// TwinCAT 3 PLC project CX2040_Project
// ProgramVersion: 3.1.4023.0
// libraries:
//   Tc2_EtherCAT, * (Beckhoff Automation GmbH)
//   Tc2_SerialCom, * (Beckhoff Automation GmbH)
//   Tc2_Standard, * (Beckhoff Automation GmbH)
//   Tc2_System, * (Beckhoff Automation GmbH)
//   Tc3_Module, * (Beckhoff Automation GmbH)
// project tree:
//   GVLs/ GVL.TcGVL
//   / PlcTask.TcTTO
//   POUs/ MAIN.TcPOU
// real-time tasks:
//   TASK PlcTask: cycle T#1ms, priority 20, ADS port 350
//   TASK PlcTask_Fast: cycle T#1ms, priority 19, ADS port 351
// I/O:
//   DEVICE Gerät 1 (EtherCAT), AmsNetId 10.183.66.136.2.1
//     Box 1 (CX2040 EtherCAT slave) [CX2040 EtherCAT slave]
// variable links:
//   CX2040 Project/CX2040 Project Instance <-> Device 1 (EtherCAT)/Box 1 (CX2040 EtherCAT slave)
//     PlcTask Inputs/MAIN.vonKlemme <-> IO Inputs/Pdo Entry 2
//     PlcTask Outputs/MAIN.test123 <-> IO Outputs/Pdo Entry 2

CONFIGURATION CX2040_Project
    RESOURCE PLC ON TwinCAT3
        TASK PlcTask(INTERVAL := T#1ms, PRIORITY := 20);
        PROGRAM MAIN WITH PlcTask : MAIN;
    END_RESOURCE
END_CONFIGURATION

// ---- GVLs/GVL.TcGVL
{attribute 'qualified_only'}
VAR_GLOBAL
	iTest AT %I* : UINT;
	NetId AT %I* : AMSNETID;
END_VAR

// ---- POUs/MAIN.TcPOU
PROGRAM MAIN
VAR
	iCount : UINT;
	fbSlaveStateChange : FB_EcSetSlaveState;
	AmsNetId : AMSNETID;
	Ams : T_AmsNetId;
	bTrigger : BOOL;
	State : WORD;
	test123 AT %Q* : USINT;
	vonKlemme AT %I* : USINT;
	
	CurrentState : ST_EcSlaveState;
END_VAR

iCount := GVL.iTest;
Ams := '10.183.66.136.4.1';
test123 := TO_USINT(iCount); 
fbSlaveStateChange(
	 sNetId := Ams,
	 nSlaveAddr := 1001,
	 bExecute := bTrigger,
	 tTimeout := T#10S,
	 reqState := State,
	 
	 bBusy =>,
	 bError =>,
	 nErrId =>,
	 currState=>
	 );
	 
CurrentState := fbSlaveStateChange.currState;

IF CurrentState.deviceState = State AND bTrigger THEN
	bTrigger := FALSE;
END_IF

END_PROGRAM
